Fanuc KAREL source: NC0080.KL

-- PROVISIONAL review KL for V770-1; original PC SHA256 dddd85ae8899edd42445131157d90780758039ae6d6ff4549fd13c562f05c40e
-- Incomplete behavior may be omitted. Consult companion uncertainty JSON. Do not deploy.
PROGRAM NC0080
%NOLOCKGROUP
-- UNRESOLVED_LOCAL_POOL 1 cells at code offset 3; source declarations unknown
-- DIRECT_LOCAL_WORD_ACCESS alone does not prove INTEGER, REAL, or BOOLEAN
BEGIN
  -- UNRESOLVED_PC offsets 0-8; opcodes 2B,2C,7B
  -- UNRESOLVED_PC offsets 13-20; opcodes 9D,23
  -- UNRESOLVED_PC offsets 25-42; opcodes 21,2E,59,79
  -- UNRESOLVED_PC offsets 47-64; opcodes 21,2E,59,79
  -- UNRESOLVED_PC offsets 69-86; opcodes 21,2E,59,79
  -- UNRESOLVED_PC offsets 91-108; opcodes 21,2E,59,79
  -- UNRESOLVED_PC offsets 113-130; opcodes 21,2E,59,79
  -- UNRESOLVED_PC offsets 135-152; opcodes 21,2E,59,79
  -- UNRESOLVED_PC offsets 157-174; opcodes 21,2E,59,79
  -- UNRESOLVED_PC offsets 179-196; opcodes 21,2E,59,79
  -- UNRESOLVED_PC offsets 201-218; opcodes 21,2E,59,79
  -- UNRESOLVED_PC offsets 223-240; opcodes 21,2E,59,79
  -- UNRESOLVED_PC offsets 245-262; opcodes 21,2E,59,79
  -- UNRESOLVED_PC offsets 267-284; opcodes 21,2E,59,79
  -- UNRESOLVED_PC offsets 289-306; opcodes 21,2E,59,79
  -- UNRESOLVED_PC offsets 311-328; opcodes 21,2E,59,79
  -- UNRESOLVED_PC offsets 333-350; opcodes 21,2E,59,79
  -- UNRESOLVED_PC offsets 355-372; opcodes 21,2E,59,79
  -- UNRESOLVED_PC offsets 377-394; opcodes 21,2E,59,79
  -- UNRESOLVED_PC offsets 399-416; opcodes 21,2E,59,79
  -- UNRESOLVED_PC offsets 421-435; opcodes 21,9D,52,23
  -- UNRESOLVED_PC offsets 440-445; opcodes 7A
  -- UNRESOLVED_PC offsets 450-455; opcodes 7A
  -- UNRESOLVED_PC offsets 460-465; opcodes 7A
  -- UNRESOLVED_PC offsets 470-475; opcodes 7A
  -- UNRESOLVED_PC offsets 480-485; opcodes 7A
  -- UNRESOLVED_PC offsets 490-495; opcodes 7A
  -- UNRESOLVED_PC offsets 500-505; opcodes 7A
  -- UNRESOLVED_PC offsets 510-515; opcodes 7A
  -- UNRESOLVED_PC offsets 520-525; opcodes 7A
  -- UNRESOLVED_PC offsets 530-535; opcodes 7A
  -- UNRESOLVED_PC offsets 540-545; opcodes 7A
  -- UNRESOLVED_PC offsets 550-555; opcodes 7A
  -- UNRESOLVED_PC offsets 560-565; opcodes 7A
  -- UNRESOLVED_PC offsets 570-575; opcodes 7A
  -- UNRESOLVED_PC offsets 580-585; opcodes 7A
  -- UNRESOLVED_PC offsets 590-595; opcodes 7A
  -- UNRESOLVED_PC offsets 600-605; opcodes 7A
  -- UNRESOLVED_PC offsets 610-615; opcodes 7A
  -- UNRESOLVED_PC offsets 620-624; opcodes 7F
  -- UNRESOLVED_PC offsets 629-633; opcodes 27,AA
  -- UNRESOLVED_PC offsets 638-642; opcodes 7F
END NC0080
